FUNCTION_BLOCK Test_RTrimEx_HandlesEmptySubject EXTENDS T_UnitTestBase
VAR_INPUT
END_VAR
VAR_OUTPUT
END_VAR
VAR
    SubjectString : T_MaxString := '';
END_VAR

METHOD Init
VAR_INPUT
END_VAR
END_METHOD

{attribute 'analysis' := '-33'} // inhibit unused variable warning
METHOD RunTest
AssertEquals_STRING(Expected := '',
                    Actual   := F_RTrimEx(n := 1, str := SubjectString),
                    Message  := 'F_LTrimEx(SubjectString)');

TestCompleted := TRUE;
END_METHOD

END_FUNCTION_BLOCK

(* stored: Version 1.1.0.1, ProductVersion 3.1.4024.12
   POU Test_RTrimEx_HandlesEmptySubject: Id {4d5e2987-0ffa-0d67-2069-2aff409ff0a5}, SpecialFunc None
   Method Init: Id {e9c11614-bbf7-0853-0e01-6c0591dc839e}
   Method RunTest: Id {2edc380c-9298-0fc8-0504-b23da452b146} *)
